// TwinCAT 3 PLC project Main
// ProgramVersion: 3.1.4023.0
// libraries:
//   Tc2_Standard, * (Beckhoff Automation GmbH)
//   Tc2_System, * (Beckhoff Automation GmbH)
//   Tc3_Module, * (Beckhoff Automation GmbH)
//   TcUnit, * (www.tcunit.org)
//   mobject-events,1.1.0,mobject
// project tree:
//   / PlcTask.TcTTO (not stored)
//   POUs/ MAIN.TcPOU
//   Tests/ EventTargetInterface_TestSuite.TcPOU, EventEmitter_TestSuite.TcPOU, EventEmitterInterface_TestSuite.TcPOU, EventHandlerInterface_TestSuite.TcPOU
//   Tests/Mocks/ MockEvent.TcPOU, MockEventHandler.TcPOU
// real-time tasks:
//   TASK PlcTask: cycle T#10ms, priority 20, ADS port 350

// ---- POUs/MAIN.TcPOU
PROGRAM MAIN
VAR
	eventEmitter_TestSuite : EventEmitter_TestSuite;
	eventEmitterInterface_TestSuite : EventEmitterInterface_TestSuite;
	eventTargetInterface_TestSuite : EventTargetInterface_TestSuite;
	eventHandlerInterface_TestSuite : EventHandlerInterface_TestSuite;
END_VAR

TcUnit.RUN();

END_PROGRAM

// ---- Tests/EventEmitter_TestSuite.TcPOU
FUNCTION_BLOCK PUBLIC EventEmitter_TestSuite EXTENDS TcUnit.FB_TestSuite
VAR
END_VAR

CheckEmitWorksWithHandler();
CheckEmitWorksWithMultipleHandlers();
CheckEventIsNotSentToTheWrongHandler();
CheckOffEventUnregistersAHandler();
CheckClearUnregistersMultipleHandlers();
CheckOnceEventCorrectlyCallsHandler();
CheckOnceEventCorrectlyCallsHandlerOnlyOnce();

METHOD PUBLIC CheckClearUnregistersMultipleHandlers
VAR
	mockEvent : MockEvent;
	mockHandler1 : MockEventHandler;
	mockHandler2 : MockEventHandler;
	eventEmitter : EventEmitter;
	eventReceived : BOOL;
END_VAR
TEST('CheckClearUnregistersMultipleHandlers');

eventEmitter.OnEvent('test', mockHandler1);
eventEmitter.OnEvent('test', mockHandler2);
eventEmitter.Clear();

eventEmitter.Emit('test',mockEvent);
eventReceived := mockHandler1.EqualsLastEvent(mockEvent) OR mockHandler2.EqualsLastEvent(mockEvent) ;

AssertFalse(
	Condition := eventReceived,
	Message := 'Event Emitter did not correctly unregister multiple handlers following a clear'
);

TEST_FINISHED();
END_METHOD

METHOD PUBLIC CheckEmitWorksWithHandler
VAR
	mockEvent : MockEvent;
	mockHandler : MockEventHandler;
	eventEmitter : EventEmitter;
	eventReceived : BOOL;
END_VAR
TEST('CheckEmitWorksWithHandler');

eventEmitter.OnEvent('test', mockHandler);

eventEmitter.Emit('test',mockEvent);
eventReceived := mockHandler.EqualsLastEvent(mockEvent);

AssertTrue(
	Condition := eventReceived,
	Message := 'Event Emitter did not correctly emmit the event to the handler'
);

TEST_FINISHED();
END_METHOD

METHOD PUBLIC CheckEmitWorksWithMultipleHandlers
VAR
	mockEvent : MockEvent;
	mockHandler1 : MockEventHandler;
	mockHandler2 : MockEventHandler;
	eventEmitter : EventEmitter;
	eventReceived : BOOL;
END_VAR
TEST('CheckEmitWorksWithMultipleHandlers');

eventEmitter.OnEvent('test', mockHandler1);
eventEmitter.OnEvent('test', mockHandler2);

eventEmitter.Emit('test',mockEvent);
eventReceived := mockHandler1.EqualsLastEvent(mockEvent) AND mockHandler2.EqualsLastEvent(mockEvent) ;

AssertTrue(
	Condition := eventReceived,
	Message := 'Event Emitter did not correctly emmit the event to multiple handlers'
);

TEST_FINISHED();
END_METHOD

METHOD PUBLIC CheckEventIsNotSentToTheWrongHandler
VAR
	mockEvent : MockEvent;
	mockHandler : MockEventHandler;
	eventEmitter : EventEmitter;
	eventReceived : BOOL;
END_VAR
TEST('CheckEventIsNotSentToTheWrongHandler');

eventEmitter.OnEvent('foo', mockHandler);

eventEmitter.Emit('bar',mockEvent);
eventReceived := mockHandler.EqualsLastEvent(mockEvent);

AssertFalse(
	Condition := eventReceived,
	Message := 'Event Emitter sent the event to the wrong handler'
);

TEST_FINISHED();
END_METHOD

METHOD PUBLIC CheckOffEventUnregistersAHandler
VAR
	mockEvent : MockEvent;
	mockHandler : MockEventHandler;
	eventEmitter : EventEmitter;
	eventReceived : BOOL;
END_VAR
TEST('CheckOffEventUnregistersAHandler');

eventEmitter.OnEvent('test', mockHandler);
eventEmitter.OffEvent('test', mockHandler);

eventEmitter.Emit('test',mockEvent);
eventReceived := mockHandler.EqualsLastEvent(mockEvent);

AssertFalse(
	Condition := eventReceived,
	Message := 'Event Emitter did not correctly unregister the event handler using the off method'
);

TEST_FINISHED();
END_METHOD

METHOD PUBLIC CheckOnceEventCorrectlyCallsHandler
VAR
	mockEvent : MockEvent;
	mockHandler : MockEventHandler;
	eventEmitter : EventEmitter;
	eventReceived : BOOL;
END_VAR
TEST('CheckOnceEventCorrectlyCallsHandler');

eventEmitter.OnceEvent('test', mockHandler);

eventEmitter.Emit('test',mockEvent);
eventReceived := mockHandler.EqualsLastEvent(mockEvent);

AssertTrue(
	Condition := eventReceived,
	Message := 'Event Emitter did not notify the handler'
);

TEST_FINISHED();
END_METHOD

METHOD PUBLIC CheckOnceEventCorrectlyCallsHandlerOnlyOnce
VAR
	mockEvent : MockEvent;
	mockHandler : MockEventHandler;
	eventEmitter : EventEmitter;
	eventCount : INT;
	expected : INT := 1;
END_VAR
TEST('CheckOnceEventCorrectlyCallsHandlerOnlyOnce');

eventEmitter.OnceEvent('test', mockHandler);

eventEmitter.Emit('test',mockEvent);
eventEmitter.Emit('test',mockEvent);
eventCount := mockHandler.EventsHandled;

AssertEquals(
	Expected := expected,
	Actual := eventCount,
	Message := 'Event Emitter notified the handler too many times'
);

TEST_FINISHED();
END_METHOD

END_FUNCTION_BLOCK

// ---- Tests/Mocks/MockEvent.TcPOU
FUNCTION_BLOCK MockEvent IMPLEMENTS I_Event
VAR
	_name : T_MAXSTRING;
END_VAR

END_FUNCTION_BLOCK

// ---- Tests/Mocks/MockEventHandler.TcPOU
FUNCTION_BLOCK MockEventHandler IMPLEMENTS I_EventHandler
VAR
	_eventsHandled : INT;
	lastEventHandled : I_Event;
END_VAR

METHOD PUBLIC EqualsLastEvent : bool
VAR_INPUT
	Event : I_Event;
END_VAR
EqualsLastEvent := lastEventHandled = Event;
END_METHOD

PROPERTY EventsHandled : int
GET
EventsHandled := _eventsHandled;
END_GET
END_PROPERTY

METHOD HandleEvent
VAR_INPUT
	Event	: I_Event;
END_VAR
_eventsHandled := _eventsHandled + 1;
lastEventHandled := Event;
END_METHOD

END_FUNCTION_BLOCK

// ---- Tests/EventEmitterInterface_TestSuite.TcPOU
FUNCTION_BLOCK PUBLIC EventEmitterInterface_TestSuite EXTENDS TcUnit.FB_TestSuite
VAR
END_VAR

CheckEmitWorksWithHandler();
CheckExtendsFromQueryInterface();
CheckOffEventUnregistersAHandler();
CheckOnceEventCorrectlyCallsHandler();

METHOD PUBLIC CheckEmitWorksWithHandler
VAR
	mockEvent : MockEvent;
	mockHandler : MockEventHandler;
	eventEmitter : EventEmitter;
	iEventEmitter : I_EventEmitter := eventEmitter;
	eventReceived : BOOL;
END_VAR
TEST('CheckEmitWorksWithHandler');

iEventEmitter.OnEvent('test', mockHandler);

eventEmitter.Emit('test',mockEvent);
eventReceived := mockHandler.EqualsLastEvent(mockEvent);

AssertTrue(
	Condition := eventReceived,
	Message := 'Event Emitter did not correctly emmit the event to the handler'
);

TEST_FINISHED();
END_METHOD

METHOD PUBLIC CheckExtendsFromQueryInterface
VAR
	eventEmitter : EventEmitter;
	iEventEmitter : I_EventEmitter := eventEmitter;
	iQueryInterface : __SYSTEM.IQueryInterface;
	result : BOOL;
END_VAR
TEST('CheckExtendsFromQueryInterface');

result := __QUERYINTERFACE(iEventEmitter,iQueryInterface);

AssertTrue(
	Condition := result,
	Message := 'Interface did not extend __SYSTEM.IQueryInterface'
);

TEST_FINISHED();
END_METHOD

METHOD PUBLIC CheckOffEventUnregistersAHandler
VAR
	mockEvent : MockEvent;
	mockHandler : MockEventHandler;
	eventEmitter : EventEmitter;
	iEventEmitter : I_EventEmitter := eventEmitter;
	eventReceived : BOOL;
END_VAR
TEST('CheckOffEventUnregistersAHandler');

iEventEmitter.OnEvent('test', mockHandler);
iEventEmitter.OffEvent('test', mockHandler);

eventEmitter.Emit('test',mockEvent);
eventReceived := mockHandler.EqualsLastEvent(mockEvent);

AssertFalse(
	Condition := eventReceived,
	Message := 'Event Emitter did not correctly unregister the event handler using the off method'
);

TEST_FINISHED();
END_METHOD

METHOD PUBLIC CheckOnceEventCorrectlyCallsHandler
VAR
	mockEvent : MockEvent;
	mockHandler : MockEventHandler;
	eventEmitter : EventEmitter;
	iEventEmitter : I_EventEmitter := eventEmitter;
	eventReceived : BOOL;
END_VAR
TEST('CheckOnceEventCorrectlyCallsHandler');

iEventEmitter.OnceEvent('test', mockHandler);

eventEmitter.Emit('test',mockEvent);
eventReceived := mockHandler.EqualsLastEvent(mockEvent);

AssertTrue(
	Condition := eventReceived,
	Message := 'Event Emitter did not notify the handler'
);

TEST_FINISHED();
END_METHOD

END_FUNCTION_BLOCK

// ---- Tests/EventTargetInterface_TestSuite.TcPOU
FUNCTION_BLOCK PUBLIC EventTargetInterface_TestSuite EXTENDS TcUnit.FB_TestSuite
VAR
END_VAR

CheckEmitWorksWithHandler();
CheckExtendsFromQueryInterface();

METHOD PUBLIC CheckEmitWorksWithHandler
VAR
	mockEvent : MockEvent;
	mockHandler : MockEventHandler;
	eventEmitter : EventEmitter;
	iEventTarget : I_EventTarget := eventEmitter;
	eventReceived : BOOL;
END_VAR
TEST('CheckEmitWorksWithHandler');

eventEmitter.OnEvent('test', mockHandler);

iEventTarget.Emit('test',mockEvent);
eventReceived := mockHandler.EqualsLastEvent(mockEvent);

AssertTrue(
	Condition := eventReceived,
	Message := 'Event Emitter did not correctly emmit the event to the handler'
);

TEST_FINISHED();
END_METHOD

METHOD PUBLIC CheckExtendsFromQueryInterface
VAR
	eventEmitter : EventEmitter;
	iEventTarget : I_EventTarget := eventEmitter;
	iQueryInterface : __SYSTEM.IQueryInterface;
	result : BOOL;
END_VAR
TEST('CheckExtendsFromQueryInterface');

result := __QUERYINTERFACE(iEventTarget,iQueryInterface);

AssertTrue(
	Condition := result,
	Message := 'Interface did not extend __SYSTEM.IQueryInterface'
);

TEST_FINISHED();
END_METHOD

END_FUNCTION_BLOCK

// ---- Tests/EventHandlerInterface_TestSuite.TcPOU
FUNCTION_BLOCK PUBLIC EventHandlerInterface_TestSuite EXTENDS TcUnit.FB_TestSuite
VAR
END_VAR

CheckEmitWorksWithHandler();
CheckExtendsFromQueryInterface();

METHOD PUBLIC CheckEmitWorksWithHandler
VAR
	mockEvent : MockEvent;
	mockHandler : MockEventHandler;
	iEventHandler : I_EventHandler := mockHandler;
	eventEmitter : EventEmitter;
	eventReceived : BOOL;
END_VAR
TEST('CheckEmitWorksWithHandler');

eventEmitter.OnEvent('test', iEventHandler);

eventEmitter.Emit('test',mockEvent);
eventReceived := mockHandler.EqualsLastEvent(mockEvent);

AssertTrue(
	Condition := eventReceived,
	Message := 'Event Emitter did not correctly emmit the event to the handler'
);

TEST_FINISHED();
END_METHOD

METHOD PUBLIC CheckExtendsFromQueryInterface
VAR
	mockHandler : MockEventHandler;
	iEventHandler : I_EventHandler := mockHandler;
	iQueryInterface : __SYSTEM.IQueryInterface;
	result : BOOL;
END_VAR
TEST('CheckExtendsFromQueryInterface');

result := __QUERYINTERFACE(iEventHandler,iQueryInterface);

AssertTrue(
	Condition := result,
	Message := 'Interface did not extend __SYSTEM.IQueryInterface'
);

TEST_FINISHED();
END_METHOD

END_FUNCTION_BLOCK
